// TwinCAT 3 PLC project M1L1_PLC
// ProgramVersion: 3.1.4020.5
// libraries:
//   LCLS General, * (SLAC)
//   lcls-twincat-motion, * (SLAC)
//   lcls-twincat-optics, * (SLAC)
//   PMPS, * (SLAC - LCLS)
//   Tc2_MC2, * (Beckhoff Automation GmbH)
//   Tc2_Standard, * (Beckhoff Automation GmbH)
//   Tc2_System, * (Beckhoff Automation GmbH)
//   Tc2_Utilities, * (Beckhoff Automation GmbH)
//   Tc3_Module, * (Beckhoff Automation GmbH)
//   TcUnit, * (www.tcunit.org)
// project tree:
//   / PlcTask.TcTTO
//   POUs/ MAIN.TcPOU
// real-time tasks:
//   TASK PlcTask: cycle T#10ms, priority 20, ADS port 350
// motion (NC):
//   TASK NC-Task 1 SAF: cycle T#2ms, priority 4, ADS port 501
//   TASK NC-Task 1 SVB: cycle T#10ms, priority 8, ADS port 511
//   AXIS Axis_Yup (id 1)
//     General: UnitName=um
//     Dynamic: Acceleration=5050, Deceleration=5050, Jerk=5100500, DelayTime=0.008
//     Velo: SlowManual=60, FastManual=90, Maximum=200
//     OtherSettings: AllowMotionCmdToSlave=true
//     encoder EncType=29
//       EncPara: ScaleFactorNumerator=1, ScaleFactorDenominator=1000, MaxCount=#xffffffff, ReferenceSystem=1
//         Inc: RefSoftSyncMask=#x0000ffff
//     drive DrvType=24
//       DrvPara: Inverse=true
//         Analog: VeloReferenz=500, ScaleFactorActTorque=0.1
//         TimeComp: TaskDelayCycles=1
//     controller CtrType=3
//       CtrPara: PriorControlFactor=1
//         PosDiffControl: Range=50, Time=0.2
//         PID: PosTn=0.005, PosIOutputLimit=0.0001, PosDOutputLimit=0, PosIDisableWhenMoving=true, DeadBandPosition=0.001
//         Observer: BandWidth=20
//   AXIS Axis_Ydwn (id 2)
//     General: UnitName=um
//     Dynamic: Acceleration=5050, Deceleration=5050, Jerk=5100500, DelayTime=0.008
//     Velo: SlowManual=60, FastManual=90, Maximum=200
//     OtherSettings: AllowMotionCmdToSlave=true
//     encoder EncType=29
//       EncPara: ScaleFactorNumerator=1, ScaleFactorDenominator=1000, MaxCount=#xffffffff, ReferenceSystem=1
//         Inc: RefSoftSyncMask=#x0000ffff
//     drive DrvType=24
//       DrvPara: Inverse=true
//         Analog: VeloReferenz=500, ScaleFactorActTorque=0.1
//         TimeComp: TaskDelayCycles=1
//     controller CtrType=3
//       CtrPara: PriorControlFactor=1
//         PosDiffControl: Range=50, Time=0.2
//         PID: PosTn=0.005, PosIOutputLimit=0.0001, PosDOutputLimit=0, PosIDisableWhenMoving=true, DeadBandPosition=0.001
//         Observer: BandWidth=20
//   AXIS Axis_Xup (id 3)
//     General: UnitName=um
//     Dynamic: Acceleration=1000, Deceleration=1000, Jerk=5000, DelayTime=0.008
//     Velo: FastManual=150, Maximum=300
//     OtherSettings: AllowMotionCmdToSlave=true
//     encoder EncType=29
//       EncPara: ScaleFactorNumerator=0.001, MaxCount=#xffffffff, ReferenceSystem=1
//         Inc: RefSoftSyncMask=#x0000ffff
//     drive DrvType=24
//       DrvPara: Inverse=true
//         Analog: VeloReferenz=625, ScaleFactorActTorque=0.1
//         TimeComp: TaskDelayCycles=1
//     controller CtrType=1
//       CtrPara: PriorControlFactor=1
//         PosDiffControl: Range=50
//         Observer: BandWidth=20
//   AXIS Axis_Xdwn (id 4)
//     General: UnitName=um
//     Dynamic: Acceleration=1000, Deceleration=1000, Jerk=5000, DelayTime=0.008
//     Velo: FastManual=150, Maximum=300
//     OtherSettings: AllowMotionCmdToSlave=true
//     encoder EncType=29
//       EncPara: ScaleFactorNumerator=0.001, MaxCount=#xffffffff, ReferenceSystem=1
//         Inc: RefSoftSyncMask=#x0000ffff
//     drive DrvType=24
//       Analog: VeloReferenz=625, ScaleFactorActTorque=0.1
//       TimeComp: TaskDelayCycles=1
//     controller CtrType=1
//       CtrPara: PriorControlFactor=1
//         PosDiffControl: Range=50
//         Observer: BandWidth=20
//   AXIS Axis_PitchCoarse (id 5)
//     General: UnitName=urad
//     Dynamic: AccelerationMaximum=7042, Acceleration=64082, Deceleration=64082, Jerk=711156, DelayTime=0.008, VeloJumpFactor=2000
//     Velo: SlowManual=30, FastManual=50, Maximum=100
//     MotionControl: Time=0.1
//     TargetPosControl: Time=2
//     OtherSettings: AllowMotionCmdToSlave=true, AllowMotionCmdToExtSetGenAxis=true, PulseDistancePos=100
//     encoder EncType=29
//       EncPara: ScaleFactorNumerator=0.00556, MaxCount=#xffffffff, ReferenceSystem=1
//         Inc: RefSoftSyncMask=#x0000ffff
//     drive DrvType=24
//       DrvPara: Inverse=true
//         Analog: VeloReferenz=7042.25
//         TimeComp: TaskDelayCycles=1
//     controller CtrType=3
//       CtrPara: PriorControlFactor=1
//         PosDiffControl: Range=10, Time=0.2
//         PID: PosKp=8, PosTn=0.0005, PosIOutputLimit=5e-005, PosDOutputLimit=0, DeadBandPosition=0.1
//         Observer: BandWidth=20
// I/O:
//   DEVICE Device 1 (EtherCAT) (disabled), AmsNetId 5.54.18.124.2.1
//     Term 1 (EK1200)
//   DEVICE Device 4 (EtherCAT), AmsNetId 5.54.18.124.5.1
//     Term 4 (EK1100) [EK1100 EtherCAT Coupler (2A E-Bus)]
//       Term 5 (EL9410) [EL9410 E-Bus Power Supplier  (Diagnostics)]
//       Term 6 (EL7047) - Yup [EL7047 1Ch. Stepper motor output stage (50V, 5A)]
//       Term 7 (EL7047) - Ydwn [EL7047 1Ch. Stepper motor output stage (50V, 5A)]
//       Term 8 (EL7047) - Xup [EL7047 1Ch. Stepper motor output stage (50V, 5A)]
//       Term 9 (EL7047) - Xdwn [EL7047 1Ch. Stepper motor output stage (50V, 5A)]
//       Term 10 (EL7047) - PitchCoarse [EL7047 1Ch. Stepper motor output stage (50V, 5A)]
//       Term 11 (EL5042) - Y [EL5042 2Ch. BiSS-C Encoder]
//       Term 12 (EL5042) - X [EL5042 2Ch. BiSS-C Encoder]
//       Term 13 (EL5042) - Pitch [EL5042 2Ch. BiSS-C Encoder]
//       Term 14 (EL6001) - PitchFine [EL6001 Interface (RS232)]
//       Term 15 (EL3054) [EL3054 4Ch. Ana. Input 4-20mA]
//       Term 16 (EL3202-0010) [EL3202-0010 2Ch. Ana. Input PT100 (RTD), High Precision]
//       Term 17 (EL3202-0010) [EL3202-0010 2Ch. Ana. Input PT100 (RTD), High Precision]
//       Term 18 (EL1004)
//       Term 19 (EL9011)
// variable links:
//   Axes/Axis_PitchCoarse <-> Device 4 (EtherCAT)/Term 4 (EK1100)/Term 10 (EL7047) - PitchCoarse
//     Drive/Inputs/In/nState1 @bit 3 <-> STM Status/Status/Error
//     Drive/Inputs/In/nState1 @bit 7 <-> STM Status/Status/Motor stall
//     Drive/Inputs/In/nState1 @bit 5 <-> STM Status/Status/Moving negative
//     Drive/Inputs/In/nState1 @bit 4 <-> STM Status/Status/Moving positive
//     Drive/Inputs/In/nState1 @bit 1 <-> STM Status/Status/Ready
//     Drive/Inputs/In/nState1 <-> STM Status/Status/Ready to enable
//     Drive/Inputs/In/nState1 @bit 6 <-> STM Status/Status/Torque reduced
//     Drive/Inputs/In/nState1 @bit 2 <-> STM Status/Status/Warning
//     Drive/Inputs/In/nState2 @bit 3 <-> STM Status/Status/Digital input 1
//     Drive/Inputs/In/nState2 @bit 4 <-> STM Status/Status/Digital input 2
//     Drive/Inputs/In/nState2 @bit 5 <-> STM Status/Status/Sync error
//     Drive/Inputs/In/nState2 @bit 7 <-> STM Status/Status/TxPDO Toggle
//     Drive/Inputs/In/nState4 @bit 1 <-> WcState/InputToggle
//     Drive/Inputs/In/nState4 <-> WcState/WcState
//     Drive/Outputs/Out/nCtrl1 <-> STM Control/Control/Enable
//     Drive/Outputs/Out/nCtrl1 @bit 2 <-> STM Control/Control/Reduce torque
//     Drive/Outputs/Out/nCtrl1 @bit 1 <-> STM Control/Control/Reset
//     Drive/Outputs/Out/nCtrl2 @bit 3 <-> STM Control/Control/Digital output 1
//     Drive/Outputs/Out/nDataOut2[0] <-> STM Velocity/Velocity
//   Axes/Axis_PitchCoarse <-> Device 4 (EtherCAT)/Term 4 (EK1100)/Term 13 (EL5042) - Pitch
//     Enc/Inputs/In/nComState @bit 1 <-> WcState/InputToggle
//     Enc/Inputs/In/nComState <-> WcState/WcState
//     Enc/Inputs/In/nDataIn1 <-> FB Inputs Channel 1/Position
//     Enc/Inputs/In/nState1 @bit 12 <-> FB Inputs Channel 1/Status/Diag
//     Enc/Inputs/In/nState1 @bit 1 <-> FB Inputs Channel 1/Status/Error
//     Enc/Inputs/In/nState1 @bit 14 <-> FB Inputs Channel 1/Status/Input cycle counter
//     Enc/Inputs/In/nState1 @bit 2 <-> FB Inputs Channel 1/Status/Ready
//     Enc/Inputs/In/nState1 @bit 13 <-> FB Inputs Channel 1/Status/TxPDO State
//     Enc/Inputs/In/nState1 <-> FB Inputs Channel 1/Status/Warning
//   Axes/Axis_Xdwn <-> Device 4 (EtherCAT)/Term 4 (EK1100)/Term 12 (EL5042) - X
//     Enc/Inputs/In/nComState @bit 1 <-> WcState/InputToggle
//     Enc/Inputs/In/nComState <-> WcState/WcState
//     Enc/Inputs/In/nDataIn1 <-> FB Inputs Channel 2/Position
//     Enc/Inputs/In/nState1 @bit 12 <-> FB Inputs Channel 2/Status/Diag
//     Enc/Inputs/In/nState1 @bit 1 <-> FB Inputs Channel 2/Status/Error
//     Enc/Inputs/In/nState1 @bit 14 <-> FB Inputs Channel 2/Status/Input cycle counter
//     Enc/Inputs/In/nState1 @bit 2 <-> FB Inputs Channel 2/Status/Ready
//     Enc/Inputs/In/nState1 @bit 13 <-> FB Inputs Channel 2/Status/TxPDO State
//     Enc/Inputs/In/nState1 <-> FB Inputs Channel 2/Status/Warning
//   Axes/Axis_Xdwn <-> Device 4 (EtherCAT)/Term 4 (EK1100)/Term 9 (EL7047) - Xdwn
//     Drive/Inputs/In/nState1 @bit 3 <-> STM Status/Status/Error
//     Drive/Inputs/In/nState1 @bit 7 <-> STM Status/Status/Motor stall
//     Drive/Inputs/In/nState1 @bit 5 <-> STM Status/Status/Moving negative
//     Drive/Inputs/In/nState1 @bit 4 <-> STM Status/Status/Moving positive
//     Drive/Inputs/In/nState1 @bit 1 <-> STM Status/Status/Ready
//     Drive/Inputs/In/nState1 <-> STM Status/Status/Ready to enable
//     Drive/Inputs/In/nState1 @bit 6 <-> STM Status/Status/Torque reduced
//     Drive/Inputs/In/nState1 @bit 2 <-> STM Status/Status/Warning
//     Drive/Inputs/In/nState2 @bit 3 <-> STM Status/Status/Digital input 1
//     Drive/Inputs/In/nState2 @bit 4 <-> STM Status/Status/Digital input 2
//     Drive/Inputs/In/nState2 @bit 5 <-> STM Status/Status/Sync error
//     Drive/Inputs/In/nState2 @bit 7 <-> STM Status/Status/TxPDO Toggle
//     Drive/Inputs/In/nState4 @bit 1 <-> WcState/InputToggle
//     Drive/Inputs/In/nState4 <-> WcState/WcState
//     Drive/Outputs/Out/nCtrl1 <-> STM Control/Control/Enable
//     Drive/Outputs/Out/nCtrl1 @bit 2 <-> STM Control/Control/Reduce torque
//     Drive/Outputs/Out/nCtrl1 @bit 1 <-> STM Control/Control/Reset
//     Drive/Outputs/Out/nCtrl2 @bit 3 <-> STM Control/Control/Digital output 1
//     Drive/Outputs/Out/nDataOut2[0] <-> STM Velocity/Velocity
//   Axes/Axis_Xup <-> Device 4 (EtherCAT)/Term 4 (EK1100)/Term 12 (EL5042) - X
//     Enc/Inputs/In/nComState @bit 1 <-> WcState/InputToggle
//     Enc/Inputs/In/nComState <-> WcState/WcState
//     Enc/Inputs/In/nDataIn1 <-> FB Inputs Channel 1/Position
//     Enc/Inputs/In/nState1 @bit 12 <-> FB Inputs Channel 1/Status/Diag
//     Enc/Inputs/In/nState1 @bit 1 <-> FB Inputs Channel 1/Status/Error
//     Enc/Inputs/In/nState1 @bit 14 <-> FB Inputs Channel 1/Status/Input cycle counter
//     Enc/Inputs/In/nState1 @bit 2 <-> FB Inputs Channel 1/Status/Ready
//     Enc/Inputs/In/nState1 @bit 13 <-> FB Inputs Channel 1/Status/TxPDO State
//     Enc/Inputs/In/nState1 <-> FB Inputs Channel 1/Status/Warning
//   Axes/Axis_Xup <-> Device 4 (EtherCAT)/Term 4 (EK1100)/Term 8 (EL7047) - Xup
//     Drive/Inputs/In/nState1 @bit 3 <-> STM Status/Status/Error
//     Drive/Inputs/In/nState1 @bit 7 <-> STM Status/Status/Motor stall
//     Drive/Inputs/In/nState1 @bit 5 <-> STM Status/Status/Moving negative
//     Drive/Inputs/In/nState1 @bit 4 <-> STM Status/Status/Moving positive
//     Drive/Inputs/In/nState1 @bit 1 <-> STM Status/Status/Ready
//     Drive/Inputs/In/nState1 <-> STM Status/Status/Ready to enable
//     Drive/Inputs/In/nState1 @bit 6 <-> STM Status/Status/Torque reduced
//     Drive/Inputs/In/nState1 @bit 2 <-> STM Status/Status/Warning
//     Drive/Inputs/In/nState2 @bit 3 <-> STM Status/Status/Digital input 1
//     Drive/Inputs/In/nState2 @bit 4 <-> STM Status/Status/Digital input 2
//     Drive/Inputs/In/nState2 @bit 5 <-> STM Status/Status/Sync error
//     Drive/Inputs/In/nState2 @bit 7 <-> STM Status/Status/TxPDO Toggle
//     Drive/Inputs/In/nState4 @bit 1 <-> WcState/InputToggle
//     Drive/Inputs/In/nState4 <-> WcState/WcState
//     Drive/Outputs/Out/nCtrl1 <-> STM Control/Control/Enable
//     Drive/Outputs/Out/nCtrl1 @bit 2 <-> STM Control/Control/Reduce torque
//     Drive/Outputs/Out/nCtrl1 @bit 1 <-> STM Control/Control/Reset
//     Drive/Outputs/Out/nCtrl2 @bit 3 <-> STM Control/Control/Digital output 1
//     Drive/Outputs/Out/nDataOut2[0] <-> STM Velocity/Velocity
//   Axes/Axis_Ydwn <-> Device 4 (EtherCAT)/Term 4 (EK1100)/Term 11 (EL5042) - Y
//     Enc/Inputs/In/nComState @bit 1 <-> WcState/InputToggle
//     Enc/Inputs/In/nComState <-> WcState/WcState
//     Enc/Inputs/In/nDataIn1 <-> FB Inputs Channel 2/Position
//     Enc/Inputs/In/nState1 @bit 12 <-> FB Inputs Channel 2/Status/Diag
//     Enc/Inputs/In/nState1 @bit 1 <-> FB Inputs Channel 2/Status/Error
//     Enc/Inputs/In/nState1 @bit 14 <-> FB Inputs Channel 2/Status/Input cycle counter
//     Enc/Inputs/In/nState1 @bit 2 <-> FB Inputs Channel 2/Status/Ready
//     Enc/Inputs/In/nState1 @bit 13 <-> FB Inputs Channel 2/Status/TxPDO State
//     Enc/Inputs/In/nState1 <-> FB Inputs Channel 2/Status/Warning
//   Axes/Axis_Ydwn <-> Device 4 (EtherCAT)/Term 4 (EK1100)/Term 7 (EL7047) - Ydwn
//     Drive/Inputs/In/nState1 @bit 3 <-> STM Status/Status/Error
//     Drive/Inputs/In/nState1 @bit 7 <-> STM Status/Status/Motor stall
//     Drive/Inputs/In/nState1 @bit 5 <-> STM Status/Status/Moving negative
//     Drive/Inputs/In/nState1 @bit 4 <-> STM Status/Status/Moving positive
//     Drive/Inputs/In/nState1 @bit 1 <-> STM Status/Status/Ready
//     Drive/Inputs/In/nState1 <-> STM Status/Status/Ready to enable
//     Drive/Inputs/In/nState1 @bit 6 <-> STM Status/Status/Torque reduced
//     Drive/Inputs/In/nState1 @bit 2 <-> STM Status/Status/Warning
//     Drive/Inputs/In/nState2 @bit 3 <-> STM Status/Status/Digital input 1
//     Drive/Inputs/In/nState2 @bit 4 <-> STM Status/Status/Digital input 2
//     Drive/Inputs/In/nState2 @bit 5 <-> STM Status/Status/Sync error
//     Drive/Inputs/In/nState2 @bit 7 <-> STM Status/Status/TxPDO Toggle
//     Drive/Inputs/In/nState4 @bit 1 <-> WcState/InputToggle
//     Drive/Inputs/In/nState4 <-> WcState/WcState
//     Drive/Outputs/Out/nCtrl1 <-> STM Control/Control/Enable
//     Drive/Outputs/Out/nCtrl1 @bit 2 <-> STM Control/Control/Reduce torque
//     Drive/Outputs/Out/nCtrl1 @bit 1 <-> STM Control/Control/Reset
//     Drive/Outputs/Out/nCtrl2 @bit 3 <-> STM Control/Control/Digital output 1
//     Drive/Outputs/Out/nDataOut2[0] <-> STM Velocity/Velocity
//   Axes/Axis_Yup <-> Device 4 (EtherCAT)/Term 4 (EK1100)/Term 11 (EL5042) - Y
//     Enc/Inputs/In/nComState @bit 1 <-> WcState/InputToggle
//     Enc/Inputs/In/nComState <-> WcState/WcState
//     Enc/Inputs/In/nDataIn1 <-> FB Inputs Channel 1/Position
//     Enc/Inputs/In/nState1 @bit 12 <-> FB Inputs Channel 1/Status/Diag
//     Enc/Inputs/In/nState1 @bit 1 <-> FB Inputs Channel 1/Status/Error
//     Enc/Inputs/In/nState1 @bit 14 <-> FB Inputs Channel 1/Status/Input cycle counter
//     Enc/Inputs/In/nState1 @bit 2 <-> FB Inputs Channel 1/Status/Ready
//     Enc/Inputs/In/nState1 @bit 13 <-> FB Inputs Channel 1/Status/TxPDO State
//     Enc/Inputs/In/nState1 <-> FB Inputs Channel 1/Status/Warning
//   Axes/Axis_Yup <-> Device 4 (EtherCAT)/Term 4 (EK1100)/Term 6 (EL7047) - Yup
//     Drive/Inputs/In/nState1 @bit 3 <-> STM Status/Status/Error
//     Drive/Inputs/In/nState1 @bit 7 <-> STM Status/Status/Motor stall
//     Drive/Inputs/In/nState1 @bit 5 <-> STM Status/Status/Moving negative
//     Drive/Inputs/In/nState1 @bit 4 <-> STM Status/Status/Moving positive
//     Drive/Inputs/In/nState1 @bit 1 <-> STM Status/Status/Ready
//     Drive/Inputs/In/nState1 <-> STM Status/Status/Ready to enable
//     Drive/Inputs/In/nState1 @bit 6 <-> STM Status/Status/Torque reduced
//     Drive/Inputs/In/nState1 @bit 2 <-> STM Status/Status/Warning
//     Drive/Inputs/In/nState2 @bit 3 <-> STM Status/Status/Digital input 1
//     Drive/Inputs/In/nState2 @bit 4 <-> STM Status/Status/Digital input 2
//     Drive/Inputs/In/nState2 @bit 5 <-> STM Status/Status/Sync error
//     Drive/Inputs/In/nState2 @bit 7 <-> STM Status/Status/TxPDO Toggle
//     Drive/Inputs/In/nState4 @bit 1 <-> WcState/InputToggle
//     Drive/Inputs/In/nState4 <-> WcState/WcState
//     Drive/Outputs/Out/nCtrl1 <-> STM Control/Control/Enable
//     Drive/Outputs/Out/nCtrl1 @bit 2 <-> STM Control/Control/Reduce torque
//     Drive/Outputs/Out/nCtrl1 @bit 1 <-> STM Control/Control/Reset
//     Drive/Outputs/Out/nCtrl2 @bit 3 <-> STM Control/Control/Digital output 1
//     Drive/Outputs/Out/nDataOut2[0] <-> STM Velocity/Velocity
//   M1L1_PLC Instance <-> Device 4 (EtherCAT)/Term 4 (EK1100)/Term 10 (EL7047) - PitchCoarse
//     PlcTask Inputs/MAIN.M5.bLimitBackwardEnable <-> STM Status/Status/Digital input 2
//     PlcTask Inputs/MAIN.M5.bLimitForwardEnable <-> STM Status/Status/Digital input 1
//   M1L1_PLC Instance <-> Device 4 (EtherCAT)/Term 4 (EK1100)/Term 11 (EL5042) - Y
//     PlcTask Inputs/MAIN.y_dwn_enc/Count <-> FB Inputs Channel 2/Position
//     PlcTask Inputs/MAIN.y_up_enc/Count <-> FB Inputs Channel 1/Position
//   M1L1_PLC Instance <-> Device 4 (EtherCAT)/Term 4 (EK1100)/Term 12 (EL5042) - X
//     PlcTask Inputs/MAIN.x_dwn_enc/Count <-> FB Inputs Channel 2/Position
//     PlcTask Inputs/MAIN.x_up_enc/Count <-> FB Inputs Channel 1/Position
//   M1L1_PLC Instance <-> Device 4 (EtherCAT)/Term 4 (EK1100)/Term 18 (EL1004)
//     PlcTask Inputs/MAIN.stoEnable1 <-> Channel 1/Input
//     PlcTask Inputs/MAIN.stoEnable2 <-> Channel 2/Input
//   M1L1_PLC Instance <-> Device 4 (EtherCAT)/Term 4 (EK1100)/Term 6 (EL7047) - Yup
//     PlcTask Inputs/MAIN.M1.bLimitBackwardEnable <-> STM Status/Status/Digital input 2
//     PlcTask Inputs/MAIN.M1.bLimitForwardEnable <-> STM Status/Status/Digital input 1
//   M1L1_PLC Instance <-> Device 4 (EtherCAT)/Term 4 (EK1100)/Term 7 (EL7047) - Ydwn
//     PlcTask Inputs/MAIN.M2.bLimitBackwardEnable <-> STM Status/Status/Digital input 2
//     PlcTask Inputs/MAIN.M2.bLimitForwardEnable <-> STM Status/Status/Digital input 1
//   M1L1_PLC Instance <-> Device 4 (EtherCAT)/Term 4 (EK1100)/Term 8 (EL7047) - Xup
//     PlcTask Inputs/MAIN.M3.bLimitBackwardEnable <-> STM Status/Status/Digital input 2
//     PlcTask Inputs/MAIN.M3.bLimitForwardEnable <-> STM Status/Status/Digital input 1
//   M1L1_PLC Instance <-> Device 4 (EtherCAT)/Term 4 (EK1100)/Term 9 (EL7047) - Xdwn
//     PlcTask Inputs/MAIN.M4.bLimitBackwardEnable <-> STM Status/Status/Digital input 2
//     PlcTask Inputs/MAIN.M4.bLimitForwardEnable <-> STM Status/Status/Digital input 1
//   M1L1_PLC Instance <-> NC-Task 1 SAF/Axes/Axis_PitchCoarse
//     PlcTask Inputs/MAIN.M5.Axis.NcToPlc <-> Outputs/ToPlc
//     PlcTask Outputs/MAIN.M5.Axis.PlcToNc <-> Inputs/FromPlc
//   M1L1_PLC Instance <-> NC-Task 1 SAF/Axes/Axis_Xdwn
//     PlcTask Inputs/MAIN.M4.Axis.NcToPlc <-> Outputs/ToPlc
//     PlcTask Outputs/MAIN.M4.Axis.PlcToNc <-> Inputs/FromPlc
//   M1L1_PLC Instance <-> NC-Task 1 SAF/Axes/Axis_Xup
//     PlcTask Inputs/MAIN.M3.Axis.NcToPlc <-> Outputs/ToPlc
//     PlcTask Outputs/MAIN.M3.Axis.PlcToNc <-> Inputs/FromPlc
//   M1L1_PLC Instance <-> NC-Task 1 SAF/Axes/Axis_Ydwn
//     PlcTask Inputs/MAIN.M2.Axis.NcToPlc <-> Outputs/ToPlc
//     PlcTask Outputs/MAIN.M2.Axis.PlcToNc <-> Inputs/FromPlc
//   M1L1_PLC Instance <-> NC-Task 1 SAF/Axes/Axis_Yup
//     PlcTask Inputs/MAIN.M1.Axis.NcToPlc <-> Outputs/ToPlc
//     PlcTask Outputs/MAIN.M1.Axis.PlcToNc <-> Inputs/FromPlc

CONFIGURATION M1L1_PLC
    RESOURCE PLC ON TwinCAT3
        TASK PlcTask(INTERVAL := T#10ms, PRIORITY := 20);
        PROGRAM MAIN WITH PlcTask : MAIN;
    END_RESOURCE
END_CONFIGURATION

// ---- POUs/MAIN.TcPOU
PROGRAM MAIN
VAR
    M1: DUT_MotionStage:=(nEnableMode:=ENUM_StageEnableMode.ALWAYS, bPowerSelf:=TRUE); // Yup
	M2: DUT_MotionStage:=(nEnableMode:=ENUM_StageEnableMode.ALWAYS, bPowerSelf:=TRUE); // Ydwn
	M3: DUT_MotionStage:=(nEnableMode:=ENUM_StageEnableMode.ALWAYS, bPowerSelf:=TRUE); // Xup
	M4: DUT_MotionStage:=(nEnableMode:=ENUM_StageEnableMode.ALWAYS, bPowerSelf:=TRUE); // Xdwn
	M5: DUT_MotionStage:=(nEnableMode:=ENUM_StageEnableMode.ALWAYS, bPowerSelf:=TRUE); // PitchCoarse

	fbMotionStage_x_up : FB_MotionStage;
    fbMotionStage_x_dwn : FB_MotionStage;
    fbMotionStage_y_up : FB_MotionStage;
    fbMotionStage_y_dwn : FB_MotionStage;
    fbMotionStage_pitch : FB_MotionStage;
	
	stoEnable1 AT %I* : BOOL;
	stoEnable2 AT %I* : BOOL;
	
	x_up_enc  AT %I*: ST_RenishawAbsEnc;
	x_dwn_enc  AT %I*: ST_RenishawAbsEnc;
	y_up_enc  AT %I*: ST_RenishawAbsEnc;
	y_dwn_enc  AT %I*: ST_RenishawAbsEnc;

	// Auto coupling function block
	fbAutoCoupleX : FB_GantryAutoCoupling;
	fbAutoCoupleY : FB_GantryAutoCoupling;
	bExecuteCoupleX : BOOL;
	bExecuteCoupleY : BOOL;
	bExecuteDecoupleX : BOOL;
	bExecuteDecoupleY : BOOL;
	bGantryAlreadyCoupledX : BOOL;
	bGantryAlreadyCoupledY : BOOL;
	
	// Gantry variables
	nCurrGantryX : LINT;
	nCurrGantryY : LINT;
	nGantryTolX : LINT := 25000;
	nGantryTolY : LINT := 25000;
END_VAR

// M1L1
// Buttons to enable motors: write 0 to enable, 2 to disable
// PitchCoarse
Main.M1.bHardwareEnable := TRUE;
fbMotionStage_y_up(stMotionStage:=Main.M1);

Main.M2.bHardwareEnable := TRUE;
fbMotionStage_y_dwn(stMotionStage:=Main.M2);

Main.M3.bHardwareEnable := TRUE;
fbMotionStage_x_up(stMotionStage:=Main.M3);

Main.M4.bHardwareEnable := TRUE;
fbMotionStage_x_dwn(stMotionStage:=Main.M4);

// Encoder Reference Values: Using Axilon FAT values
y_up_enc.Ref := 108558460;
y_dwn_enc.Ref := 108761210;
x_up_enc.Ref := 20664670; 
x_dwn_enc.Ref := 20133000;

// Gantry Differences to monitor
nCurrGantryY := ((ULINT_TO_LINT(y_up_enc.Count) - ULINT_TO_LINT(y_up_enc.Ref)) - (ULINT_TO_LINT(y_dwn_enc.Count) - ULINT_TO_LINT(y_dwn_enc.Ref)));
nCurrGantryX := ((ULINT_TO_LINT(x_up_enc.Count) - ULINT_TO_LINT(x_up_enc.Ref)) - (ULINT_TO_LINT(x_dwn_enc.Count) - ULINT_TO_LINT(x_dwn_enc.Ref)));

// E-stop
M1.bHardwareEnable := stoEnable1 AND stoEnable2;
M2.bHardwareEnable := stoEnable1 AND stoEnable2;
M3.bHardwareEnable := stoEnable1 AND stoEnable2;
M4.bHardwareEnable := stoEnable1 AND stoEnable2;
M5.bHardwareEnable := stoEnable1 AND stoEnable2;


// Start Autocoupling
fbAutoCoupleX(nGantryTol:=nGantryTolX, Master:=M3, MasterEnc:=x_up_enc, Slave:=M4,
	          SlaveEnc:=x_dwn_enc, bExecuteCouple:=bExecuteCoupleX,
              bExecuteDecouple:=bExecuteDecoupleX,
              bGantryAlreadyCoupled=>bGantryAlreadyCoupledX);

fbAutoCoupleY(nGantryTol:=nGantryTolY, Master:=M1, MasterEnc:=y_up_enc, Slave:=M2,
	          SlaveEnc:=y_dwn_enc, bExecuteCouple:=bExecuteCoupleY,
              bExecuteDecouple:=bExecuteDecoupleY,
			  bGantryAlreadyCoupled=>bGantryAlreadyCoupledY);

fbMotionStage_y_up  (stMotionStage:=M1);
fbMotionStage_y_dwn (stMotionStage:=M2);
fbMotionStage_x_up  (stMotionStage:=M3);
fbMotionStage_x_dwn (stMotionStage:=M4);
fbMotionStage_pitch (stMotionStage:=M5);

END_PROGRAM
